RESOURCE_TYPE top_evstation
  (* Standard: 61499-2 *)
  (* Version 0.1, 2018-00-07, hpea485, UOA *)
  FBS
    inputs : sifb_bfb_inputs;
    Reference1 : print;
    battery : bfb_ess_battery;
    controller : cfb_controller;
    Reference : bfb_text_print;
  END_FBS
  EVENT_CONNECTIONS
    inputs.Tick TO controller.Tick;
    inputs.Tick TO Reference.tick_stop;
    Reference1.Done TO Reference.Tick_array;
    battery.SoC_change TO Reference1.Last_Tick;
    battery.SoC_change TO Reference.Tick_SoC;
    battery.Discharge_out TO Reference1.Discharging;
    battery.Charge_out TO Reference1.Charging;
    battery.Do_nothing_out TO Reference1.Do_nothing;
    controller.Charging TO battery.Charge;
    controller.Discharging TO battery.Discharge;
    controller.Do_nothing TO battery.Do_nothing;
    controller.Tick_time TO battery.Tick_ESS;
    Reference.Done TO inputs.Start;
  END_CONNECTIONS
  DATA_CONNECTIONS
    inputs.Minute TO controller.Minute;
    inputs.Minute TO Reference1.Minute;
    inputs.Price TO controller.Price;
    inputs.Price TO Reference1.Price;
    inputs.Demand_kWh TO controller.Demand_kWh;
    inputs.Day TO controller.day;
    inputs.Day TO Reference.Day;
    inputs.Lenght TO Reference.lenght;
    inputs.stop TO Reference.Stop;
    inputs.Sma TO controller.Sma;
    inputs.Sma TO Reference.SMA;
    inputs.Std_dev TO controller.Std_dev;
    inputs.Std_dev TO Reference.Std_dev;
    Reference1.min TO Reference.Min;
    Reference1.Demand TO Reference.Demand;
    Reference1.Pgrid TO Reference.Pgrid;
    Reference1.Pbc TO Reference.Pbc;
    Reference1.Pbd TO Reference.Pbd;
    Reference1.Price_min TO Reference.Price;
    battery.BatterySoC TO controller.ESS_battery_SoC;
    battery.BatterySoC TO Reference.SoC;
    battery.Demand TO Reference1.Power_Demand;
    controller.ESS_Charging_Power_Demand TO battery.Charge_Power;
    controller.ESS_Charging_Power_Demand TO Reference1.ESS_Charging;
    controller.ESS_Discharging_Power TO battery.Discharge_Power;
    controller.ESS_Discharging_Power TO Reference1.ESS_Discharging_Power;
    controller.SoC TO battery.SoC_input;
    controller.Demand TO battery.Power_Demand;
  END_CONNECTIONS
END_RESOURCE_TYPE
